# EPICS substitutions: kstar/siteApp/TS1/TS1App/Db/ts_value_B1.substitutions
#
file db/TS_CH_value.db
{
    pattern
        { DEV,    ID,       TAIL,     DESC,                ARG     }

        {"B1",    "0",      "VALUE",   "raw value",    "raw_cur"}
        {"B1",    "1",       "VALUE",   "raw value",    "raw_cur"}
        {"B1",    "2",       "VALUE",   "raw value",    "raw_cur"}
        {"B1",    "3",       "VALUE",   "raw value",    "raw_cur"}
        {"B1",    "4",       "VALUE",   "raw value",    "raw_cur"}
        {"B1",    "5",       "VALUE",   "raw value",    "raw_cur"}
        {"B1",    "6",       "VALUE",   "raw value",    "raw_cur"}
        {"B1",    "7",       "VALUE",   "raw value",    "raw_cur"}
        {"B1",    "8",       "VALUE",   "raw value",    "raw_cur"}
        {"B1",    "9",       "VALUE",   "raw value",    "raw_cur"}
        {"B1",    "10",       "VALUE",   "raw value",    "raw_cur"}
        {"B1",    "11",       "VALUE",   "raw value",    "raw_cur"}
        {"B1",    "12",       "VALUE",   "raw value",    "raw_cur"}
        {"B1",    "13",       "VALUE",   "raw value",    "raw_cur"}
        {"B1",    "14",       "VALUE",   "raw value",    "raw_cur"}
        {"B1",    "15",       "VALUE",   "raw value",    "raw_cur"}
        {"B1",    "16",       "VALUE",   "raw value",    "raw_cur"}
        {"B1",    "17",       "VALUE",   "raw value",    "raw_cur"}
        {"B1",    "18",       "VALUE",   "raw value",    "raw_cur"}
        {"B1",    "19",       "VALUE",   "raw value",    "raw_cur"}
        {"B1",    "20",       "VALUE",   "raw value",    "raw_cur"}
        {"B1",    "21",       "VALUE",   "raw value",    "raw_cur"}
        {"B1",    "22",       "VALUE",   "raw value",    "raw_cur"}
        {"B1",    "23",       "VALUE",   "raw value",    "raw_cur"}
        {"B1",    "24",       "VALUE",   "raw value",    "raw_cur"}
        {"B1",    "25",       "VALUE",   "raw value",    "raw_cur"}
        {"B1",    "26",       "VALUE",   "raw value",    "raw_cur"}
        {"B1",    "27",       "VALUE",   "raw value",    "raw_cur"}
        {"B1",    "28",       "VALUE",   "raw value",    "raw_cur"}
        {"B1",    "29",       "VALUE",   "raw value",    "raw_cur"}
        {"B1",    "30",       "VALUE",   "raw value",    "raw_cur"}
        {"B1",    "31",       "VALUE",   "raw value",    "raw_cur"}

}
